(* IEC 61131-3 sources: virtuepot/watertank/openplc-program, 3 files *)

(* ---- simple-control.st ---- *)
PROGRAM Hello_World
  VAR
    level AT %IW101 : UINT;
    outflow AT %QW100 : UINT;
  END_VAR
  VAR
    max_level : REAL := 1200.0;
    min_level : REAL := 800.0;
    convert_to_level : REAL := 32.768;
    convert_from_flow : REAL := 1638.4;
    low_flow : REAL := 15.0;
    high_flow : REAL := 25.0;
    UINT_TO_REAL3_OUT : REAL;
    DIV10_OUT : REAL;
    GT11_OUT : BOOL;
    LT13_OUT : BOOL;
    SEL16_OUT : REAL;
    SEL15_OUT : REAL;
    MUL8_OUT : REAL;
    REAL_TO_UINT4_OUT : UINT;
  END_VAR

  UINT_TO_REAL3_OUT := UINT_TO_REAL(level);
  DIV10_OUT := DIV(UINT_TO_REAL3_OUT, convert_to_level);
  GT11_OUT := GT(DIV10_OUT, max_level);
  LT13_OUT := LT(DIV10_OUT, min_level);
  SEL16_OUT := SEL(LT13_OUT, SEL15_OUT, low_flow);
  SEL15_OUT := SEL(GT11_OUT, SEL16_OUT, high_flow);
  MUL8_OUT := MUL(SEL15_OUT, convert_from_flow);
  REAL_TO_UINT4_OUT := REAL_TO_UINT(MUL8_OUT);
  outflow := REAL_TO_UINT4_OUT;
END_PROGRAM

CONFIGURATION Config0

  RESOURCE Res0 ON PLC
    TASK task0(INTERVAL := T#300ms,PRIORITY := 0);
    PROGRAM instance0 WITH task0 : Hello_World;
  END_RESOURCE
END_CONFIGURATION

(* ---- simple-control3.st ---- *)
PROGRAM Hello_World
  VAR
    level AT %IW101 : UINT;
    outflow AT %QW100 : UINT;
    max_level AT %QW1 : UINT := 1200;
    min_level AT %QW2 : UINT := 800;
  END_VAR
  VAR
    convert_to_level : REAL := 32.768;
    convert_from_flow : REAL := 1638.4;
    low_flow : REAL := 15.0;
    high_flow : REAL := 25.0;
    UINT_TO_REAL3_OUT : REAL;
    DIV10_OUT : REAL;
    UINT_TO_REAL6_OUT : REAL;
    GT11_OUT : BOOL;
    UINT_TO_REAL9_OUT : REAL;
    LT13_OUT : BOOL;
    SEL16_OUT : REAL;
    SEL15_OUT : REAL;
    MUL8_OUT : REAL;
    REAL_TO_UINT4_OUT : UINT;
  END_VAR

  UINT_TO_REAL3_OUT := UINT_TO_REAL(level);
  DIV10_OUT := DIV(UINT_TO_REAL3_OUT, convert_to_level);
  UINT_TO_REAL6_OUT := UINT_TO_REAL(max_level);
  GT11_OUT := GT(DIV10_OUT, UINT_TO_REAL6_OUT);
  UINT_TO_REAL9_OUT := UINT_TO_REAL(min_level);
  LT13_OUT := LT(DIV10_OUT, UINT_TO_REAL9_OUT);
  SEL16_OUT := SEL(LT13_OUT, SEL15_OUT, low_flow);
  SEL15_OUT := SEL(GT11_OUT, SEL16_OUT, high_flow);
  MUL8_OUT := MUL(SEL15_OUT, convert_from_flow);
  REAL_TO_UINT4_OUT := REAL_TO_UINT(MUL8_OUT);
  outflow := REAL_TO_UINT4_OUT;
END_PROGRAM

CONFIGURATION Config0

  RESOURCE Res0 ON PLC
    TASK task0(INTERVAL := T#300ms,PRIORITY := 0);
    PROGRAM instance0 WITH task0 : Hello_World;
  END_RESOURCE
END_CONFIGURATION

(* ---- watertank.st ---- *)
PROGRAM water_tank
VAR
  level: REAL;
  areal: REAL;
  height: REAL;
  inflow: REAL;
  inflow_mean: REAL;
  inflow_stddev: REAL;
  max_inflow: REAL;
  outflow: REAL;
  max_outflow: REAL;
  set_level: REAL;
END_VAR

  level := 1000.0;
  areal := 1000000.0;
  height := 2000.0;
  inflow := 20.0;
  inflow_mean := 20.0;
  inflow_stddev := 3.0;
  max_inflow := 40.0;
  outflow := 20.0;
  max_outflow := 40.0;
  set_level := 1000.0;

  WHILE (TRUE) DO
    inflow := inflow_mean + (RANDOM - 0.5) * inflow_stddev;
    IF (inflow > max_inflow) THEN
      inflow := max_inflow;
    END_IF;

    level := level + inflow - outflow;

    IF (level > height) THEN
      level := height;
    END_IF;

    IF (level < 0) THEN
      level := 0;
    END_IF;

    outflow := (level - set_level) * areal;

    IF (outflow > max_outflow) THEN
      outflow := max_outflow;
    END_IF;
  END_WHILE;
END_PROGRAM
